FUNCTION Convert_STRING_TO_LREAL : BOOL
VAR_INPUT
	in : STRING;
	out : REFERENCE TO LREAL;
END_VAR
VAR
	converted : LREAL;
END_VAR

converted := STRING_TO_LREAL(in);

IF (LREAL_TO_STRING(converted) <> in) THEN
	RETURN;
END_IF

out := converted;
Convert_STRING_TO_LREAL := TRUE;

END_FUNCTION

(* stored: Version 1.1.0.1, ProductVersion 3.1.4024.12
   POU Convert_STRING_TO_LREAL: Id {5751001e-2116-4a7e-bb42-b75ebb07de38}, SpecialFunc None *)
